// LS Electric XG5000 project: 동남-39
// PLC NewPLC
// module base 0 slot 0: 입출력 모듈:XBC-DN/DP14E (DC 24V 입력 8점, 트랜지스터 출력 6점)

PROGRAM NewProgram (task: 스캔 프로그램)

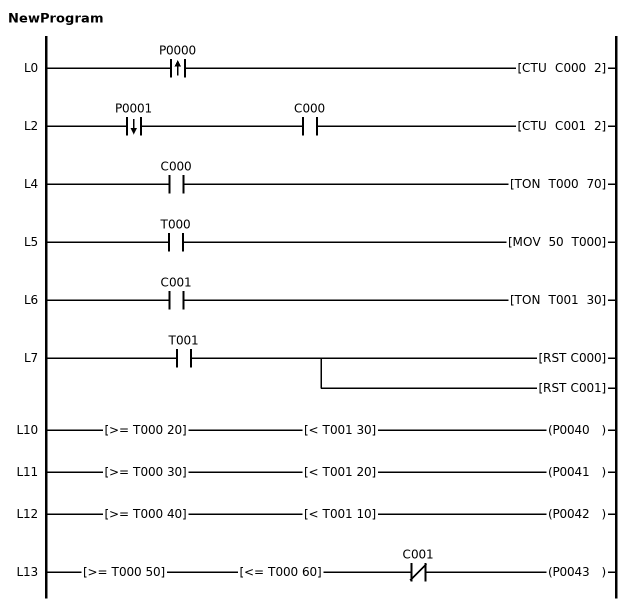
; L0
LOADP     P0000
CTU       C000 2
; L2
LOADN     P0001
AND       C000
CTU       C001 2
; L4
LOAD      C000
TON       T000 70
; L5
LOAD      T000
MOV       50 T000
; L6
LOAD      C001
TON       T001 30
; L7
LOAD      T001
RST       C000
RST       C001
; L10
LOAD>=    T000 20
AND<      T001 30
OUT       P0040
; L11
LOAD>=    T000 30
AND<      T001 20
OUT       P0041
; L12
LOAD>=    T000 40
AND<      T001 10
OUT       P0042
; L13
LOAD>=    T000 50
AND<=     T000 60
AND NOT   C001
OUT       P0043